// TIA Portal V18 export
FUNCTION "TIME CONV" : Void   // FC3, LAD
{ S7_Optimized_Access := 'TRUE' }
VERSION : 0.1
// stored: AutoNumber true, IsIECCheckEnabled false, SetENOAutomatically false, UDAEnableTagReadback false
   VAR_INPUT
      MODE : Bool;
   END_VAR
   VAR_IN_OUT
      MIN : Int;
      SEC : Int;
      "TIME" : Time;
   END_VAR
   VAR_TEMP
      "MUL VAL" : DInt;
   END_VAR
BEGIN

REGION Network 1 (SCL)
   IF #MODE THEN
       #"MUL VAL" := INT_TO_DINT(#SEC + #MIN*60);
       #"MUL VAL" := #"MUL VAL" * 1000;
       #TIME := DINT_TO_TIME( #"MUL VAL");
   ELSIF NOT #MODE THEN
       //nokkanda unni ith njan alla
       #MIN := DINT_TO_INT(((TIME_TO_DINT(#TIME) /1000)/60));
       #SEC := DINT_TO_INT(((TIME_TO_DINT(#TIME)/ 1000 MOD 60)));
   END_IF;
END_REGION
END_FUNCTION
